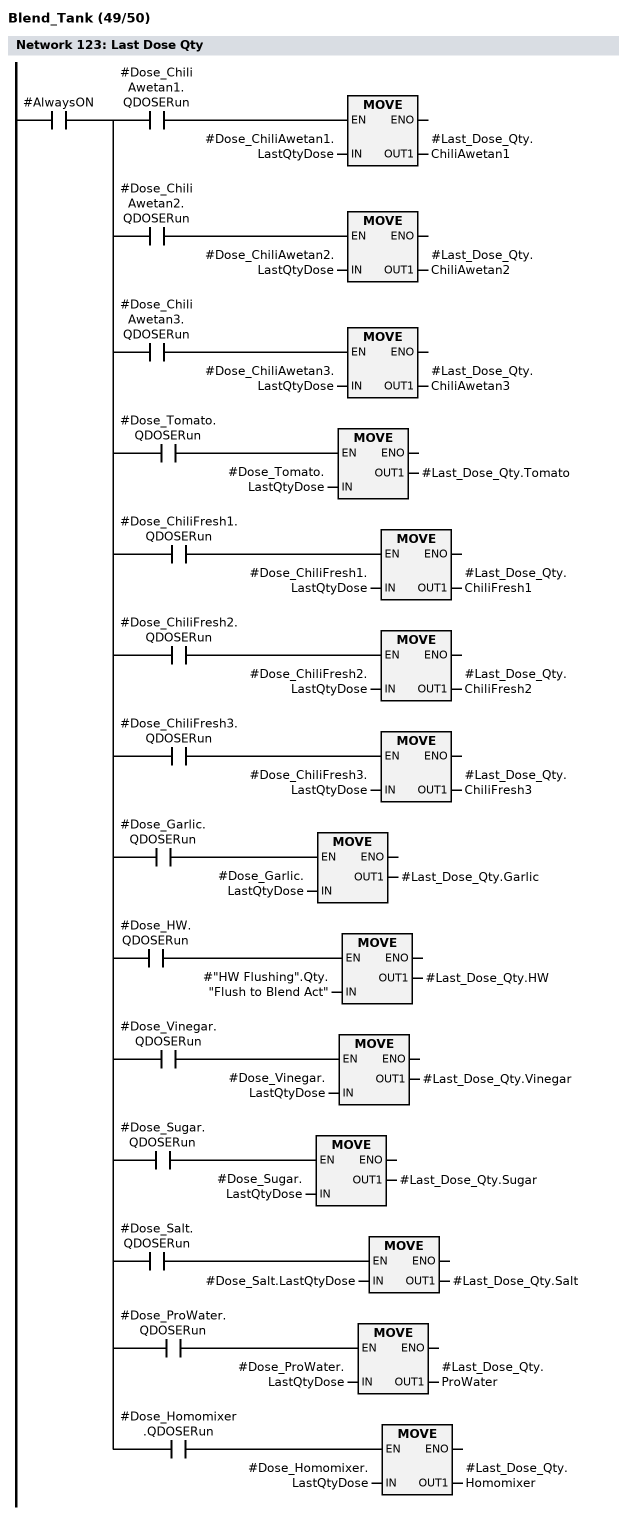
   RUNG wire#powerrail
      Contact( #AlwaysON )
      wire#w1
      Contact( #Dose_ChiliAwetan1.QDOSERun )
      Move(in := #Dose_ChiliAwetan1.LastQtyDose, out1 => #Last_Dose_Qty.ChiliAwetan1)
   END_RUNG
   RUNG wire#w1
      Contact( #Dose_ChiliAwetan2.QDOSERun )
      Move(in := #Dose_ChiliAwetan2.LastQtyDose, out1 => #Last_Dose_Qty.ChiliAwetan2)
   END_RUNG
   RUNG wire#w1
      Contact( #Dose_ChiliAwetan3.QDOSERun )
      Move(in := #Dose_ChiliAwetan3.LastQtyDose, out1 => #Last_Dose_Qty.ChiliAwetan3)
   END_RUNG
   RUNG wire#w1
      Contact( #Dose_Tomato.QDOSERun )
      Move(in := #Dose_Tomato.LastQtyDose, out1 => #Last_Dose_Qty.Tomato)
   END_RUNG
   RUNG wire#w1
      Contact( #Dose_ChiliFresh1.QDOSERun )
      Move(in := #Dose_ChiliFresh1.LastQtyDose, out1 => #Last_Dose_Qty.ChiliFresh1)
   END_RUNG
   RUNG wire#w1
      Contact( #Dose_ChiliFresh2.QDOSERun )
      Move(in := #Dose_ChiliFresh2.LastQtyDose, out1 => #Last_Dose_Qty.ChiliFresh2)
   END_RUNG
   RUNG wire#w1
      Contact( #Dose_ChiliFresh3.QDOSERun )
      Move(in := #Dose_ChiliFresh3.LastQtyDose, out1 => #Last_Dose_Qty.ChiliFresh3)
   END_RUNG
   RUNG wire#w1
      Contact( #Dose_Garlic.QDOSERun )
      Move(in := #Dose_Garlic.LastQtyDose, out1 => #Last_Dose_Qty.Garlic)
   END_RUNG
   RUNG wire#w1
      Contact( #Dose_HW.QDOSERun )
      Move(in := #"HW Flushing".Qty."Flush to Blend Act", out1 => #Last_Dose_Qty.HW)
   END_RUNG
   RUNG wire#w1
      Contact( #Dose_Vinegar.QDOSERun )
      Move(in := #Dose_Vinegar.LastQtyDose, out1 => #Last_Dose_Qty.Vinegar)
   END_RUNG
   RUNG wire#w1
      Contact( #Dose_Sugar.QDOSERun )
      Move(in := #Dose_Sugar.LastQtyDose, out1 => #Last_Dose_Qty.Sugar)
   END_RUNG
   RUNG wire#w1
      Contact( #Dose_Salt.QDOSERun )
      Move(in := #Dose_Salt.LastQtyDose, out1 => #Last_Dose_Qty.Salt)
   END_RUNG
   RUNG wire#w1
      Contact( #Dose_ProWater.QDOSERun )
      Move(in := #Dose_ProWater.LastQtyDose, out1 => #Last_Dose_Qty.ProWater)
   END_RUNG
   RUNG wire#w1
      Contact( #Dose_Homomixer.QDOSERun )
      Move(in := #Dose_Homomixer.LastQtyDose, out1 => #Last_Dose_Qty.Homomixer)
   END_RUNG
   // the same network as SCL:
   IF #AlwaysON AND #Dose_ChiliAwetan1.QDOSERun THEN
       #Last_Dose_Qty.ChiliAwetan1 := #Dose_ChiliAwetan1.LastQtyDose;
   END_IF;
   IF #AlwaysON AND #Dose_ChiliAwetan2.QDOSERun THEN
       #Last_Dose_Qty.ChiliAwetan2 := #Dose_ChiliAwetan2.LastQtyDose;
   END_IF;
   IF #AlwaysON AND #Dose_ChiliAwetan3.QDOSERun THEN
       #Last_Dose_Qty.ChiliAwetan3 := #Dose_ChiliAwetan3.LastQtyDose;
   END_IF;
   IF #AlwaysON AND #Dose_Tomato.QDOSERun THEN #Last_Dose_Qty.Tomato := #Dose_Tomato.LastQtyDose; END_IF;
   IF #AlwaysON AND #Dose_ChiliFresh1.QDOSERun THEN
       #Last_Dose_Qty.ChiliFresh1 := #Dose_ChiliFresh1.LastQtyDose;
   END_IF;
   IF #AlwaysON AND #Dose_ChiliFresh2.QDOSERun THEN
       #Last_Dose_Qty.ChiliFresh2 := #Dose_ChiliFresh2.LastQtyDose;
   END_IF;
   IF #AlwaysON AND #Dose_ChiliFresh3.QDOSERun THEN
       #Last_Dose_Qty.ChiliFresh3 := #Dose_ChiliFresh3.LastQtyDose;
   END_IF;
   IF #AlwaysON AND #Dose_Garlic.QDOSERun THEN #Last_Dose_Qty.Garlic := #Dose_Garlic.LastQtyDose; END_IF;
   IF #AlwaysON AND #Dose_HW.QDOSERun THEN
       #Last_Dose_Qty.HW := #"HW Flushing".Qty."Flush to Blend Act";
   END_IF;
   IF #AlwaysON AND #Dose_Vinegar.QDOSERun THEN #Last_Dose_Qty.Vinegar := #Dose_Vinegar.LastQtyDose; END_IF;
   IF #AlwaysON AND #Dose_Sugar.QDOSERun THEN #Last_Dose_Qty.Sugar := #Dose_Sugar.LastQtyDose; END_IF;
   IF #AlwaysON AND #Dose_Salt.QDOSERun THEN #Last_Dose_Qty.Salt := #Dose_Salt.LastQtyDose; END_IF;
   IF #AlwaysON AND #Dose_ProWater.QDOSERun THEN
       #Last_Dose_Qty.ProWater := #Dose_ProWater.LastQtyDose;
   END_IF;
   IF #AlwaysON AND #Dose_Homomixer.QDOSERun THEN
       #Last_Dose_Qty.Homomixer := #Dose_Homomixer.LastQtyDose;
   END_IF;
END_REGION

REGION Network 124: Reset Last Dose Qty After CIP Tank
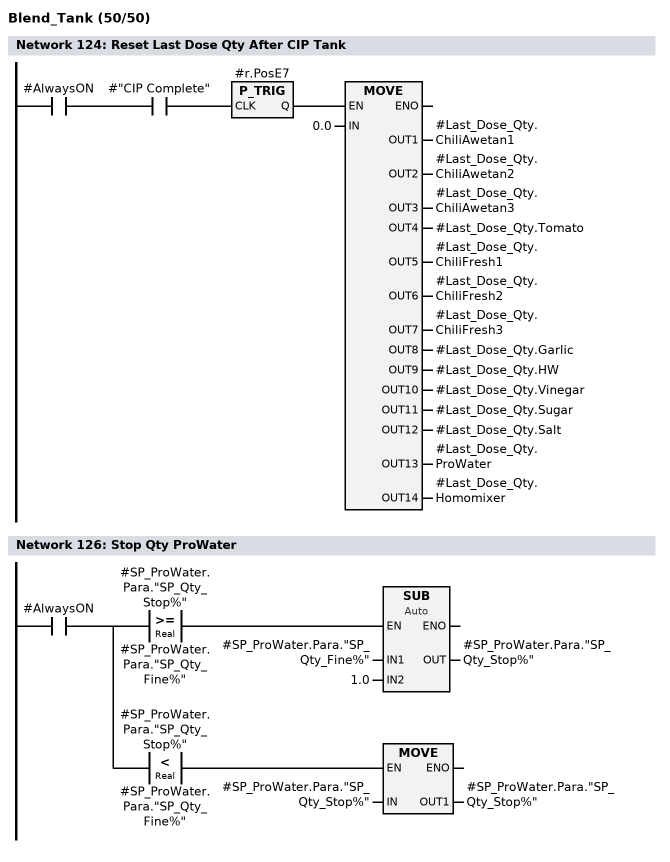
   RUNG wire#powerrail
      Contact( #AlwaysON )
      Contact( #"CIP Complete" )
      P_Trig( #r.PosE7 )
      Move(in := 0.0, out1 => #Last_Dose_Qty.ChiliAwetan1, out2 => #Last_Dose_Qty.ChiliAwetan2, out3 => #Last_Dose_Qty.ChiliAwetan3, out4 => #Last_Dose_Qty.Tomato, out5 => #Last_Dose_Qty.ChiliFresh1, out6 => #Last_Dose_Qty.ChiliFresh2, out7 => #Last_Dose_Qty.ChiliFresh3, out8 => #Last_Dose_Qty.Garlic, out9 => #Last_Dose_Qty.HW, out10 => #Last_Dose_Qty.Vinegar, out11 => #Last_Dose_Qty.Sugar, out12 => #Last_Dose_Qty.Salt, out13 => #Last_Dose_Qty.ProWater, out14 => #Last_Dose_Qty.Homomixer)
   END_RUNG
   // the same network as SCL:
   #_w1 := #AlwaysON AND #"CIP Complete";
   #_w2 := #_w1 AND NOT #r.PosE7;   // rising edge
   #r.PosE7 := #_w1;
   IF #_w2 THEN
       #Last_Dose_Qty.ChiliAwetan1 := 0.0;
       #Last_Dose_Qty.ChiliAwetan2 := 0.0;
       #Last_Dose_Qty.ChiliAwetan3 := 0.0;
       #Last_Dose_Qty.Tomato := 0.0;
       #Last_Dose_Qty.ChiliFresh1 := 0.0;
       #Last_Dose_Qty.ChiliFresh2 := 0.0;
       #Last_Dose_Qty.ChiliFresh3 := 0.0;
       #Last_Dose_Qty.Garlic := 0.0;
       #Last_Dose_Qty.HW := 0.0;
       #Last_Dose_Qty.Vinegar := 0.0;
       #Last_Dose_Qty.Sugar := 0.0;
       #Last_Dose_Qty.Salt := 0.0;
       #Last_Dose_Qty.ProWater := 0.0;
       #Last_Dose_Qty.Homomixer := 0.0;
   END_IF;
END_REGION

REGION Network 126: Stop Qty ProWater
   RUNG wire#powerrail
      Contact( #AlwaysON )
      wire#w1
      { S7_Templates := "SrcType := Real" } GE_Contact(in1 := #SP_ProWater.Para."SP_Qty_Stop%", in2 := #SP_ProWater.Para."SP_Qty_Fine%")
      Sub(in1 := #SP_ProWater.Para."SP_Qty_Fine%", in2 := 1.0, out => #SP_ProWater.Para."SP_Qty_Stop%")
   END_RUNG
   RUNG wire#w1
      { S7_Templates := "SrcType := Real" } LT_Contact(in1 := #SP_ProWater.Para."SP_Qty_Stop%", in2 := #SP_ProWater.Para."SP_Qty_Fine%")
      Move(in := #SP_ProWater.Para."SP_Qty_Stop%", out1 => #SP_ProWater.Para."SP_Qty_Stop%")
   END_RUNG
   // the same network as SCL:
   IF #AlwaysON AND (#SP_ProWater.Para."SP_Qty_Stop%" >= #SP_ProWater.Para."SP_Qty_Fine%") THEN
       #SP_ProWater.Para."SP_Qty_Stop%" := #SP_ProWater.Para."SP_Qty_Fine%" - 1.0;
   END_IF;
   IF #AlwaysON AND (#SP_ProWater.Para."SP_Qty_Stop%" < #SP_ProWater.Para."SP_Qty_Fine%") THEN
       #SP_ProWater.Para."SP_Qty_Stop%" := #SP_ProWater.Para."SP_Qty_Stop%";
   END_IF;
END_REGION
END_FUNCTION_BLOCK
